(* IEC 61131-3 sources: TIA2AX/tests/test_projects/expected/HW_1516_reader/6A1, 6 files *)

(* ---- HwInputs.st ---- *)
TYPE
	HwInputs : STRUCT
		_6A1_6A2 AT %B1000 : DWORD;
		_6A1_6A3 AT %B1004 : ARRAY[0..31] OF BYTE;
		_10A1_Acquisition_Status_1 AT %B300 : ARRAY[0..2] OF BYTE;
		_10A1_Results_Status_1 AT %B303 : BYTE;
		_10A1_Soft_Event_Control_1 AT %B304 : BYTE;
		_10A1_Result_Data_64_bytes_1 AT %B310 : ARRAY[0..71] OF BYTE;
		_11A1_11A2 AT %B100 : BYTE;
		_11A1_11A3 AT %B101 : BYTE;
		_12A1_12A2 AT %B1100 : BYTE;
		_12A1_12A3 AT %B1101 : BYTE;
	END_STRUCT;
END_TYPE

(* ---- HwOutputs.st ---- *)
TYPE
	HwOutputs : STRUCT
		_6A1_6A4 AT %B1000 : ARRAY[0..7] OF BYTE;
		_10A1_Acquisition_Control_1 AT %B300 : BYTE;
		_10A1_Results_Control_1 AT %B303 : BYTE;
		_10A1_Soft_Event_Control_1 AT %B304 : BYTE;
		_10A1_User_Data_64_bytes_1 AT %B310 : ARRAY[0..67] OF BYTE;
		_11A1_11A4 AT %B100 : BYTE;
		_12A1_12A4 AT %B1100 : WORD;
	END_STRUCT;
END_TYPE

(* ---- PlcInputs.st ---- *)
TYPE
	PlcInputs : STRUCT
		_6A1_6A2 : DWORD;
		_6A1_6A3 : ARRAY[0..31] OF BYTE;
		_10A1_Acquisition_Status_1 : ARRAY[0..2] OF BYTE;
		_10A1_Results_Status_1 : BYTE;
		_10A1_Soft_Event_Control_1 : BYTE;
		_10A1_Result_Data_64_bytes_1 : ARRAY[0..71] OF BYTE;
		_11A1_11A2 : BYTE;
		_11A1_11A3 : BYTE;
		_12A1_12A2 : BYTE;
		_12A1_12A3 : BYTE;
	END_STRUCT;
END_TYPE

(* ---- PlcOutputs.st ---- *)
TYPE
	PlcOutputs : STRUCT
		_6A1_6A4 : ARRAY[0..7] OF BYTE;
		_10A1_Acquisition_Control_1 : BYTE;
		_10A1_Results_Control_1 : BYTE;
		_10A1_Soft_Event_Control_1 : BYTE;
		_10A1_User_Data_64_bytes_1 : ARRAY[0..67] OF BYTE;
		_11A1_11A4 : BYTE;
		_12A1_12A4 : WORD;
	END_STRUCT;
END_TYPE

(* ---- CopyInputs.st ---- *)
FUNCTION CopyInputs
	VAR_EXTERNAL
		HwInputs : HwInputs;
		PlcInputs : PlcInputs;
	END_VAR
	PlcInputs._6A1_6A2 := HwInputs._6A1_6A2;
	PlcInputs._6A1_6A3[0] := HwInputs._6A1_6A3[0];
	PlcInputs._6A1_6A3[1] := HwInputs._6A1_6A3[1];
	PlcInputs._6A1_6A3[2] := HwInputs._6A1_6A3[2];
	PlcInputs._6A1_6A3[3] := HwInputs._6A1_6A3[3];
	PlcInputs._6A1_6A3[4] := HwInputs._6A1_6A3[4];
	PlcInputs._6A1_6A3[5] := HwInputs._6A1_6A3[5];
	PlcInputs._6A1_6A3[6] := HwInputs._6A1_6A3[6];
	PlcInputs._6A1_6A3[7] := HwInputs._6A1_6A3[7];
	PlcInputs._6A1_6A3[8] := HwInputs._6A1_6A3[8];
	PlcInputs._6A1_6A3[9] := HwInputs._6A1_6A3[9];
	PlcInputs._6A1_6A3[10] := HwInputs._6A1_6A3[10];
	PlcInputs._6A1_6A3[11] := HwInputs._6A1_6A3[11];
	PlcInputs._6A1_6A3[12] := HwInputs._6A1_6A3[12];
	PlcInputs._6A1_6A3[13] := HwInputs._6A1_6A3[13];
	PlcInputs._6A1_6A3[14] := HwInputs._6A1_6A3[14];
	PlcInputs._6A1_6A3[15] := HwInputs._6A1_6A3[15];
	PlcInputs._6A1_6A3[16] := HwInputs._6A1_6A3[16];
	PlcInputs._6A1_6A3[17] := HwInputs._6A1_6A3[17];
	PlcInputs._6A1_6A3[18] := HwInputs._6A1_6A3[18];
	PlcInputs._6A1_6A3[19] := HwInputs._6A1_6A3[19];
	PlcInputs._6A1_6A3[20] := HwInputs._6A1_6A3[20];
	PlcInputs._6A1_6A3[21] := HwInputs._6A1_6A3[21];
	PlcInputs._6A1_6A3[22] := HwInputs._6A1_6A3[22];
	PlcInputs._6A1_6A3[23] := HwInputs._6A1_6A3[23];
	PlcInputs._6A1_6A3[24] := HwInputs._6A1_6A3[24];
	PlcInputs._6A1_6A3[25] := HwInputs._6A1_6A3[25];
	PlcInputs._6A1_6A3[26] := HwInputs._6A1_6A3[26];
	PlcInputs._6A1_6A3[27] := HwInputs._6A1_6A3[27];
	PlcInputs._6A1_6A3[28] := HwInputs._6A1_6A3[28];
	PlcInputs._6A1_6A3[29] := HwInputs._6A1_6A3[29];
	PlcInputs._6A1_6A3[30] := HwInputs._6A1_6A3[30];
	PlcInputs._6A1_6A3[31] := HwInputs._6A1_6A3[31];
	PlcInputs._10A1_Acquisition_Status_1[0] := HwInputs._10A1_Acquisition_Status_1[0];
	PlcInputs._10A1_Acquisition_Status_1[1] := HwInputs._10A1_Acquisition_Status_1[1];
	PlcInputs._10A1_Acquisition_Status_1[2] := HwInputs._10A1_Acquisition_Status_1[2];
	PlcInputs._10A1_Results_Status_1 := HwInputs._10A1_Results_Status_1;
	PlcInputs._10A1_Soft_Event_Control_1 := HwInputs._10A1_Soft_Event_Control_1;
	PlcInputs._10A1_Result_Data_64_bytes_1[0] := HwInputs._10A1_Result_Data_64_bytes_1[0];
	PlcInputs._10A1_Result_Data_64_bytes_1[1] := HwInputs._10A1_Result_Data_64_bytes_1[1];
	PlcInputs._10A1_Result_Data_64_bytes_1[2] := HwInputs._10A1_Result_Data_64_bytes_1[2];
	PlcInputs._10A1_Result_Data_64_bytes_1[3] := HwInputs._10A1_Result_Data_64_bytes_1[3];
	PlcInputs._10A1_Result_Data_64_bytes_1[4] := HwInputs._10A1_Result_Data_64_bytes_1[4];
	PlcInputs._10A1_Result_Data_64_bytes_1[5] := HwInputs._10A1_Result_Data_64_bytes_1[5];
	PlcInputs._10A1_Result_Data_64_bytes_1[6] := HwInputs._10A1_Result_Data_64_bytes_1[6];
	PlcInputs._10A1_Result_Data_64_bytes_1[7] := HwInputs._10A1_Result_Data_64_bytes_1[7];
	PlcInputs._10A1_Result_Data_64_bytes_1[8] := HwInputs._10A1_Result_Data_64_bytes_1[8];
	PlcInputs._10A1_Result_Data_64_bytes_1[9] := HwInputs._10A1_Result_Data_64_bytes_1[9];
	PlcInputs._10A1_Result_Data_64_bytes_1[10] := HwInputs._10A1_Result_Data_64_bytes_1[10];
	PlcInputs._10A1_Result_Data_64_bytes_1[11] := HwInputs._10A1_Result_Data_64_bytes_1[11];
	PlcInputs._10A1_Result_Data_64_bytes_1[12] := HwInputs._10A1_Result_Data_64_bytes_1[12];
	PlcInputs._10A1_Result_Data_64_bytes_1[13] := HwInputs._10A1_Result_Data_64_bytes_1[13];
	PlcInputs._10A1_Result_Data_64_bytes_1[14] := HwInputs._10A1_Result_Data_64_bytes_1[14];
	PlcInputs._10A1_Result_Data_64_bytes_1[15] := HwInputs._10A1_Result_Data_64_bytes_1[15];
	PlcInputs._10A1_Result_Data_64_bytes_1[16] := HwInputs._10A1_Result_Data_64_bytes_1[16];
	PlcInputs._10A1_Result_Data_64_bytes_1[17] := HwInputs._10A1_Result_Data_64_bytes_1[17];
	PlcInputs._10A1_Result_Data_64_bytes_1[18] := HwInputs._10A1_Result_Data_64_bytes_1[18];
	PlcInputs._10A1_Result_Data_64_bytes_1[19] := HwInputs._10A1_Result_Data_64_bytes_1[19];
	PlcInputs._10A1_Result_Data_64_bytes_1[20] := HwInputs._10A1_Result_Data_64_bytes_1[20];
	PlcInputs._10A1_Result_Data_64_bytes_1[21] := HwInputs._10A1_Result_Data_64_bytes_1[21];
	PlcInputs._10A1_Result_Data_64_bytes_1[22] := HwInputs._10A1_Result_Data_64_bytes_1[22];
	PlcInputs._10A1_Result_Data_64_bytes_1[23] := HwInputs._10A1_Result_Data_64_bytes_1[23];
	PlcInputs._10A1_Result_Data_64_bytes_1[24] := HwInputs._10A1_Result_Data_64_bytes_1[24];
	PlcInputs._10A1_Result_Data_64_bytes_1[25] := HwInputs._10A1_Result_Data_64_bytes_1[25];
	PlcInputs._10A1_Result_Data_64_bytes_1[26] := HwInputs._10A1_Result_Data_64_bytes_1[26];
	PlcInputs._10A1_Result_Data_64_bytes_1[27] := HwInputs._10A1_Result_Data_64_bytes_1[27];
	PlcInputs._10A1_Result_Data_64_bytes_1[28] := HwInputs._10A1_Result_Data_64_bytes_1[28];
	PlcInputs._10A1_Result_Data_64_bytes_1[29] := HwInputs._10A1_Result_Data_64_bytes_1[29];
	PlcInputs._10A1_Result_Data_64_bytes_1[30] := HwInputs._10A1_Result_Data_64_bytes_1[30];
	PlcInputs._10A1_Result_Data_64_bytes_1[31] := HwInputs._10A1_Result_Data_64_bytes_1[31];
	PlcInputs._10A1_Result_Data_64_bytes_1[32] := HwInputs._10A1_Result_Data_64_bytes_1[32];
	PlcInputs._10A1_Result_Data_64_bytes_1[33] := HwInputs._10A1_Result_Data_64_bytes_1[33];
	PlcInputs._10A1_Result_Data_64_bytes_1[34] := HwInputs._10A1_Result_Data_64_bytes_1[34];
	PlcInputs._10A1_Result_Data_64_bytes_1[35] := HwInputs._10A1_Result_Data_64_bytes_1[35];
	PlcInputs._10A1_Result_Data_64_bytes_1[36] := HwInputs._10A1_Result_Data_64_bytes_1[36];
	PlcInputs._10A1_Result_Data_64_bytes_1[37] := HwInputs._10A1_Result_Data_64_bytes_1[37];
	PlcInputs._10A1_Result_Data_64_bytes_1[38] := HwInputs._10A1_Result_Data_64_bytes_1[38];
	PlcInputs._10A1_Result_Data_64_bytes_1[39] := HwInputs._10A1_Result_Data_64_bytes_1[39];
	PlcInputs._10A1_Result_Data_64_bytes_1[40] := HwInputs._10A1_Result_Data_64_bytes_1[40];
	PlcInputs._10A1_Result_Data_64_bytes_1[41] := HwInputs._10A1_Result_Data_64_bytes_1[41];
	PlcInputs._10A1_Result_Data_64_bytes_1[42] := HwInputs._10A1_Result_Data_64_bytes_1[42];
	PlcInputs._10A1_Result_Data_64_bytes_1[43] := HwInputs._10A1_Result_Data_64_bytes_1[43];
	PlcInputs._10A1_Result_Data_64_bytes_1[44] := HwInputs._10A1_Result_Data_64_bytes_1[44];
	PlcInputs._10A1_Result_Data_64_bytes_1[45] := HwInputs._10A1_Result_Data_64_bytes_1[45];
	PlcInputs._10A1_Result_Data_64_bytes_1[46] := HwInputs._10A1_Result_Data_64_bytes_1[46];
	PlcInputs._10A1_Result_Data_64_bytes_1[47] := HwInputs._10A1_Result_Data_64_bytes_1[47];
	PlcInputs._10A1_Result_Data_64_bytes_1[48] := HwInputs._10A1_Result_Data_64_bytes_1[48];
	PlcInputs._10A1_Result_Data_64_bytes_1[49] := HwInputs._10A1_Result_Data_64_bytes_1[49];
	PlcInputs._10A1_Result_Data_64_bytes_1[50] := HwInputs._10A1_Result_Data_64_bytes_1[50];
	PlcInputs._10A1_Result_Data_64_bytes_1[51] := HwInputs._10A1_Result_Data_64_bytes_1[51];
	PlcInputs._10A1_Result_Data_64_bytes_1[52] := HwInputs._10A1_Result_Data_64_bytes_1[52];
	PlcInputs._10A1_Result_Data_64_bytes_1[53] := HwInputs._10A1_Result_Data_64_bytes_1[53];
	PlcInputs._10A1_Result_Data_64_bytes_1[54] := HwInputs._10A1_Result_Data_64_bytes_1[54];
	PlcInputs._10A1_Result_Data_64_bytes_1[55] := HwInputs._10A1_Result_Data_64_bytes_1[55];
	PlcInputs._10A1_Result_Data_64_bytes_1[56] := HwInputs._10A1_Result_Data_64_bytes_1[56];
	PlcInputs._10A1_Result_Data_64_bytes_1[57] := HwInputs._10A1_Result_Data_64_bytes_1[57];
	PlcInputs._10A1_Result_Data_64_bytes_1[58] := HwInputs._10A1_Result_Data_64_bytes_1[58];
	PlcInputs._10A1_Result_Data_64_bytes_1[59] := HwInputs._10A1_Result_Data_64_bytes_1[59];
	PlcInputs._10A1_Result_Data_64_bytes_1[60] := HwInputs._10A1_Result_Data_64_bytes_1[60];
	PlcInputs._10A1_Result_Data_64_bytes_1[61] := HwInputs._10A1_Result_Data_64_bytes_1[61];
	PlcInputs._10A1_Result_Data_64_bytes_1[62] := HwInputs._10A1_Result_Data_64_bytes_1[62];
	PlcInputs._10A1_Result_Data_64_bytes_1[63] := HwInputs._10A1_Result_Data_64_bytes_1[63];
	PlcInputs._10A1_Result_Data_64_bytes_1[64] := HwInputs._10A1_Result_Data_64_bytes_1[64];
	PlcInputs._10A1_Result_Data_64_bytes_1[65] := HwInputs._10A1_Result_Data_64_bytes_1[65];
	PlcInputs._10A1_Result_Data_64_bytes_1[66] := HwInputs._10A1_Result_Data_64_bytes_1[66];
	PlcInputs._10A1_Result_Data_64_bytes_1[67] := HwInputs._10A1_Result_Data_64_bytes_1[67];
	PlcInputs._10A1_Result_Data_64_bytes_1[68] := HwInputs._10A1_Result_Data_64_bytes_1[68];
	PlcInputs._10A1_Result_Data_64_bytes_1[69] := HwInputs._10A1_Result_Data_64_bytes_1[69];
	PlcInputs._10A1_Result_Data_64_bytes_1[70] := HwInputs._10A1_Result_Data_64_bytes_1[70];
	PlcInputs._10A1_Result_Data_64_bytes_1[71] := HwInputs._10A1_Result_Data_64_bytes_1[71];
	PlcInputs._11A1_11A2 := HwInputs._11A1_11A2;
	PlcInputs._11A1_11A3 := HwInputs._11A1_11A3;
	PlcInputs._12A1_12A2 := HwInputs._12A1_12A2;
	PlcInputs._12A1_12A3 := HwInputs._12A1_12A3;
END_FUNCTION

(* ---- CopyOutputs.st ---- *)
FUNCTION CopyOutputs
	VAR_EXTERNAL
		HwOutputs : HwOutputs;
		PlcOutputs : PlcOutputs;
	END_VAR
	HwOutputs._6A1_6A4[0] := PlcOutputs._6A1_6A4[0];
	HwOutputs._6A1_6A4[1] := PlcOutputs._6A1_6A4[1];
	HwOutputs._6A1_6A4[2] := PlcOutputs._6A1_6A4[2];
	HwOutputs._6A1_6A4[3] := PlcOutputs._6A1_6A4[3];
	HwOutputs._6A1_6A4[4] := PlcOutputs._6A1_6A4[4];
	HwOutputs._6A1_6A4[5] := PlcOutputs._6A1_6A4[5];
	HwOutputs._6A1_6A4[6] := PlcOutputs._6A1_6A4[6];
	HwOutputs._6A1_6A4[7] := PlcOutputs._6A1_6A4[7];
	HwOutputs._10A1_Acquisition_Control_1 := PlcOutputs._10A1_Acquisition_Control_1;
	HwOutputs._10A1_Results_Control_1 := PlcOutputs._10A1_Results_Control_1;
	HwOutputs._10A1_Soft_Event_Control_1 := PlcOutputs._10A1_Soft_Event_Control_1;
	HwOutputs._10A1_User_Data_64_bytes_1[0] := PlcOutputs._10A1_User_Data_64_bytes_1[0];
	HwOutputs._10A1_User_Data_64_bytes_1[1] := PlcOutputs._10A1_User_Data_64_bytes_1[1];
	HwOutputs._10A1_User_Data_64_bytes_1[2] := PlcOutputs._10A1_User_Data_64_bytes_1[2];
	HwOutputs._10A1_User_Data_64_bytes_1[3] := PlcOutputs._10A1_User_Data_64_bytes_1[3];
	HwOutputs._10A1_User_Data_64_bytes_1[4] := PlcOutputs._10A1_User_Data_64_bytes_1[4];
	HwOutputs._10A1_User_Data_64_bytes_1[5] := PlcOutputs._10A1_User_Data_64_bytes_1[5];
	HwOutputs._10A1_User_Data_64_bytes_1[6] := PlcOutputs._10A1_User_Data_64_bytes_1[6];
	HwOutputs._10A1_User_Data_64_bytes_1[7] := PlcOutputs._10A1_User_Data_64_bytes_1[7];
	HwOutputs._10A1_User_Data_64_bytes_1[8] := PlcOutputs._10A1_User_Data_64_bytes_1[8];
	HwOutputs._10A1_User_Data_64_bytes_1[9] := PlcOutputs._10A1_User_Data_64_bytes_1[9];
	HwOutputs._10A1_User_Data_64_bytes_1[10] := PlcOutputs._10A1_User_Data_64_bytes_1[10];
	HwOutputs._10A1_User_Data_64_bytes_1[11] := PlcOutputs._10A1_User_Data_64_bytes_1[11];
	HwOutputs._10A1_User_Data_64_bytes_1[12] := PlcOutputs._10A1_User_Data_64_bytes_1[12];
	HwOutputs._10A1_User_Data_64_bytes_1[13] := PlcOutputs._10A1_User_Data_64_bytes_1[13];
	HwOutputs._10A1_User_Data_64_bytes_1[14] := PlcOutputs._10A1_User_Data_64_bytes_1[14];
	HwOutputs._10A1_User_Data_64_bytes_1[15] := PlcOutputs._10A1_User_Data_64_bytes_1[15];
	HwOutputs._10A1_User_Data_64_bytes_1[16] := PlcOutputs._10A1_User_Data_64_bytes_1[16];
	HwOutputs._10A1_User_Data_64_bytes_1[17] := PlcOutputs._10A1_User_Data_64_bytes_1[17];
	HwOutputs._10A1_User_Data_64_bytes_1[18] := PlcOutputs._10A1_User_Data_64_bytes_1[18];
	HwOutputs._10A1_User_Data_64_bytes_1[19] := PlcOutputs._10A1_User_Data_64_bytes_1[19];
	HwOutputs._10A1_User_Data_64_bytes_1[20] := PlcOutputs._10A1_User_Data_64_bytes_1[20];
	HwOutputs._10A1_User_Data_64_bytes_1[21] := PlcOutputs._10A1_User_Data_64_bytes_1[21];
	HwOutputs._10A1_User_Data_64_bytes_1[22] := PlcOutputs._10A1_User_Data_64_bytes_1[22];
	HwOutputs._10A1_User_Data_64_bytes_1[23] := PlcOutputs._10A1_User_Data_64_bytes_1[23];
	HwOutputs._10A1_User_Data_64_bytes_1[24] := PlcOutputs._10A1_User_Data_64_bytes_1[24];
	HwOutputs._10A1_User_Data_64_bytes_1[25] := PlcOutputs._10A1_User_Data_64_bytes_1[25];
	HwOutputs._10A1_User_Data_64_bytes_1[26] := PlcOutputs._10A1_User_Data_64_bytes_1[26];
	HwOutputs._10A1_User_Data_64_bytes_1[27] := PlcOutputs._10A1_User_Data_64_bytes_1[27];
	HwOutputs._10A1_User_Data_64_bytes_1[28] := PlcOutputs._10A1_User_Data_64_bytes_1[28];
	HwOutputs._10A1_User_Data_64_bytes_1[29] := PlcOutputs._10A1_User_Data_64_bytes_1[29];
	HwOutputs._10A1_User_Data_64_bytes_1[30] := PlcOutputs._10A1_User_Data_64_bytes_1[30];
	HwOutputs._10A1_User_Data_64_bytes_1[31] := PlcOutputs._10A1_User_Data_64_bytes_1[31];
	HwOutputs._10A1_User_Data_64_bytes_1[32] := PlcOutputs._10A1_User_Data_64_bytes_1[32];
	HwOutputs._10A1_User_Data_64_bytes_1[33] := PlcOutputs._10A1_User_Data_64_bytes_1[33];
	HwOutputs._10A1_User_Data_64_bytes_1[34] := PlcOutputs._10A1_User_Data_64_bytes_1[34];
	HwOutputs._10A1_User_Data_64_bytes_1[35] := PlcOutputs._10A1_User_Data_64_bytes_1[35];
	HwOutputs._10A1_User_Data_64_bytes_1[36] := PlcOutputs._10A1_User_Data_64_bytes_1[36];
	HwOutputs._10A1_User_Data_64_bytes_1[37] := PlcOutputs._10A1_User_Data_64_bytes_1[37];
	HwOutputs._10A1_User_Data_64_bytes_1[38] := PlcOutputs._10A1_User_Data_64_bytes_1[38];
	HwOutputs._10A1_User_Data_64_bytes_1[39] := PlcOutputs._10A1_User_Data_64_bytes_1[39];
	HwOutputs._10A1_User_Data_64_bytes_1[40] := PlcOutputs._10A1_User_Data_64_bytes_1[40];
	HwOutputs._10A1_User_Data_64_bytes_1[41] := PlcOutputs._10A1_User_Data_64_bytes_1[41];
	HwOutputs._10A1_User_Data_64_bytes_1[42] := PlcOutputs._10A1_User_Data_64_bytes_1[42];
	HwOutputs._10A1_User_Data_64_bytes_1[43] := PlcOutputs._10A1_User_Data_64_bytes_1[43];
	HwOutputs._10A1_User_Data_64_bytes_1[44] := PlcOutputs._10A1_User_Data_64_bytes_1[44];
	HwOutputs._10A1_User_Data_64_bytes_1[45] := PlcOutputs._10A1_User_Data_64_bytes_1[45];
	HwOutputs._10A1_User_Data_64_bytes_1[46] := PlcOutputs._10A1_User_Data_64_bytes_1[46];
	HwOutputs._10A1_User_Data_64_bytes_1[47] := PlcOutputs._10A1_User_Data_64_bytes_1[47];
	HwOutputs._10A1_User_Data_64_bytes_1[48] := PlcOutputs._10A1_User_Data_64_bytes_1[48];
	HwOutputs._10A1_User_Data_64_bytes_1[49] := PlcOutputs._10A1_User_Data_64_bytes_1[49];
	HwOutputs._10A1_User_Data_64_bytes_1[50] := PlcOutputs._10A1_User_Data_64_bytes_1[50];
	HwOutputs._10A1_User_Data_64_bytes_1[51] := PlcOutputs._10A1_User_Data_64_bytes_1[51];
	HwOutputs._10A1_User_Data_64_bytes_1[52] := PlcOutputs._10A1_User_Data_64_bytes_1[52];
	HwOutputs._10A1_User_Data_64_bytes_1[53] := PlcOutputs._10A1_User_Data_64_bytes_1[53];
	HwOutputs._10A1_User_Data_64_bytes_1[54] := PlcOutputs._10A1_User_Data_64_bytes_1[54];
	HwOutputs._10A1_User_Data_64_bytes_1[55] := PlcOutputs._10A1_User_Data_64_bytes_1[55];
	HwOutputs._10A1_User_Data_64_bytes_1[56] := PlcOutputs._10A1_User_Data_64_bytes_1[56];
	HwOutputs._10A1_User_Data_64_bytes_1[57] := PlcOutputs._10A1_User_Data_64_bytes_1[57];
	HwOutputs._10A1_User_Data_64_bytes_1[58] := PlcOutputs._10A1_User_Data_64_bytes_1[58];
	HwOutputs._10A1_User_Data_64_bytes_1[59] := PlcOutputs._10A1_User_Data_64_bytes_1[59];
	HwOutputs._10A1_User_Data_64_bytes_1[60] := PlcOutputs._10A1_User_Data_64_bytes_1[60];
	HwOutputs._10A1_User_Data_64_bytes_1[61] := PlcOutputs._10A1_User_Data_64_bytes_1[61];
	HwOutputs._10A1_User_Data_64_bytes_1[62] := PlcOutputs._10A1_User_Data_64_bytes_1[62];
	HwOutputs._10A1_User_Data_64_bytes_1[63] := PlcOutputs._10A1_User_Data_64_bytes_1[63];
	HwOutputs._10A1_User_Data_64_bytes_1[64] := PlcOutputs._10A1_User_Data_64_bytes_1[64];
	HwOutputs._10A1_User_Data_64_bytes_1[65] := PlcOutputs._10A1_User_Data_64_bytes_1[65];
	HwOutputs._10A1_User_Data_64_bytes_1[66] := PlcOutputs._10A1_User_Data_64_bytes_1[66];
	HwOutputs._10A1_User_Data_64_bytes_1[67] := PlcOutputs._10A1_User_Data_64_bytes_1[67];
	HwOutputs._11A1_11A4 := PlcOutputs._11A1_11A4;
	HwOutputs._12A1_12A4 := PlcOutputs._12A1_12A4;
END_FUNCTION
